{attribute 'qualified_only' := ''}
{attribute 'strict' := ''}
TYPE cResolvedDBStatusRoute :
(
	None := 0,
	Empty_NoRoute := 1,
	Empty_RoutedThisStation := 2,
	Empty_RoutedOtherStation := 3,
	Normal_RoutedThisStation := 5,
	Normal_RoutedOtherStation := 6,
	Normal_RoutedException := 7,
	Normal_RoutedConsolidation := 8,
	NonNormal_RoutedException := 9,
	UnknownDevice := 10,
	FastReceivingVision := 11,
	InvalidCombination := 12
) DINT;
END_TYPE

(* stored: Version 1.1.0.1, ProductVersion 3.1.4024.6
   DUT cResolvedDBStatusRoute: Id {11782a1e-a3b4-40e6-ae99-e7c36700d0fc} *)
